FUNCTION_BLOCK INTERNAL VelocityStep2 
VAR
  tf, a0, af, vd : LREAL;
  aMax, aMin, jMax : LREAL;
END_VAR

METHOD CheckAll : BOOL
VAR_IN_OUT
  Profile : ProfileDesc;
END_VAR
VAR_INPUT
  aMax, aMin, jMax : LREAL;
END_VAR
CheckAll := time_acc0(Profile, aMax, aMin, jMax) OR_ELSE time_none(Profile, aMax, aMin, jMax);
END_METHOD

METHOD Get : BOOL
VAR_IN_OUT
  Profile : ProfileDesc;
END_VAR
// Test all cases to get ones that match
// However we should guess which one is correct and try them first...
IF (vd > 0) THEN
  Get := CheckAll(Profile, aMax, aMin, jMax) OR_ELSE CheckAll(Profile, aMin, aMax, -jMax);
ELSE
  Get := CheckAll(Profile, aMin, aMax, -jMax) OR_ELSE CheckAll(Profile, aMax, aMin, jMax);
END_IF
END_METHOD

METHOD Set
VAR_INPUT
  tf : LREAL;
  v0, a0 : LREAL;
  vf, af : LREAL;
  aMax, aMin : LREAL;
  jMax : LREAL; 
END_VAR
THIS^.a0 := a0;
THIS^.tf := tf;
THIS^.af := af;
THIS^.aMax := aMax;
THIS^.aMin := aMin;
THIS^.jMax := jMax;
THIS^.vd := vf - v0;
END_METHOD

METHOD PRIVATE time_acc0 : BOOL
VAR_IN_OUT
  profile : ProfileDesc;
END_VAR
VAR_INPUT
  aMax, aMin, jMax : LREAL;
END_VAR
VAR
  h1 : LREAL;
END_VAR
// UD Solution 1/2
h1 := (-a0*a0 - af*af + 2*a0*af + 2*jMax*((a0 + af)*tf - 2*(vd)))/(jMax*jMax) + tf*tf;
IF h1 >= 0
THEN
  h1 := SQRT(h1);
  
  profile.t[0] := (af - a0)/(2*jMax) + (tf - h1)/2;
  profile.t[1] := h1;
  profile.t[2] := tf - (profile.t[0] + h1);
  profile.t[3] := 0;
  profile.t[4] := 0;
  profile.t[5] := 0;
  profile.t[6] := 0;
  
  IF (profile.CheckForVelocity(ProfileJerkSigns.uddu, ReachedLimits.Acc0, jMax, aMax, aMin)) THEN
    profile.pf := profile.p[7];
    time_acc0 := TRUE;
    RETURN;
  END_IF
END_IF

// UU Solution
h1 := (a0 - af + jMax*tf);

profile.t[0] := -Power2(af - a0)/(2*jMax*h1) + (vd - a0*tf)/h1;
profile.t[1] := (a0 - af)/jMax + tf;
profile.t[2] := 0;
profile.t[3] := 0;
profile.t[4] := tf - (profile.t[0] + profile.t[1]);
profile.t[5] := 0;
profile.t[6] := 0;

IF (profile.CheckForVelocity(ProfileJerkSigns.udud, ReachedLimits.Acc0, jMax, aMax, aMin))
THEN
  profile.pf := profile.p[7];
  time_acc0 := TRUE;
  RETURN;
END_IF

// UU Solution - 2 step
profile.t[0] := 0;
profile.t[1] := (a0 - af)/jMax + tf;
profile.t[2] := 0;
profile.t[3] := 0;
profile.t[4] := (af - a0)/jMax;
profile.t[5] := 0;
profile.t[6] := 0;

IF (profile.CheckForVelocity(ProfileJerkSigns.udud, ReachedLimits.Acc0, jMax, aMax, aMin))
THEN
  profile.pf := profile.p[7];
  time_acc0 := TRUE;
  RETURN;
END_IF
END_METHOD

METHOD PRIVATE time_none : BOOL
VAR_IN_OUT
  profile : ProfileDesc;
END_VAR
VAR_INPUT
  aMax, aMin, jMax : LREAL;
END_VAR
VAR
  h1, jf : LREAL;
END_VAR
IF (ABS(a0) < Constants.DoubleEpsilon AND_THEN ABS(af) < Constants.DoubleEpsilon AND_THEN ABS(vd) < Constants.DoubleEpsilon) THEN
  profile.t[0] := 0;
  profile.t[1] := tf;
  profile.t[2] := 0;
  profile.t[3] := 0;
  profile.t[4] := 0;
  profile.t[5] := 0;
  profile.t[6] := 0;
  
  IF (profile.CheckForVelocity(ProfileJerkSigns.uddu, ReachedLimits.None, jMax, aMax, aMin)) THEN
    profile.pf := profile.p[7];
    time_none := TRUE;
    RETURN;
  END_IF
END_IF
    
// UD Solution 1/2
IF ABS(af - a0) > Constants.DoubleEpsilon
THEN
  h1 := 2*(af*tf - vd);
  profile.t[0] := h1/(af - a0);
  profile.t[1] := tf - profile.t[0];
  profile.t[2] := 0;
  profile.t[3] := 0;
  profile.t[4] := 0;
  profile.t[5] := 0;
  profile.t[6] := 0;
  
  jf := Power2(a0 - af)/h1;
  IF (ABS(jf) < ABS(jMax) + 1E-12 AND_THEN profile.CheckForVelocity(ProfileJerkSigns.uddu, ReachedLimits.None, jf, aMax, aMin))
  THEN
    profile.pf := profile.p[7];
    time_none := TRUE;
  END_IF
END_IF
END_METHOD

END_FUNCTION_BLOCK

(* stored: Version 1.1.0.1
   POU VelocityStep2: Id {44d0404d-f840-43a5-b935-c3fca779d43d}, SpecialFunc None
   Method CheckAll: Id {5edd91ed-f446-4dff-95cf-42bfd1ecd2c0}
   Method Get: Id {291bf2c1-3902-431e-bdad-f5b9a8de3521}
   Method Set: Id {1ea081ff-38e9-4265-a71e-f22d7dc2ecbe}
   Method time_acc0: Id {139ae830-064a-498c-9553-ea8f79b368be}
   Method time_none: Id {b7252407-1ffc-4203-89cb-177864a2876c} *)
